{attribute 'pack_mode' := '1'}
TYPE TprodCounter :
STRUCT
	dTotal		:DWORD;
	dGood		:DWORD;
END_STRUCT
END_TYPE

(* stored: Version 1.1.0.1, ProductVersion 3.1.4022.12
   DUT TprodCounter: Id {fa45f757-f6e3-4ec4-a483-842dc93c3bf8} *)
